FUNCTION_BLOCK FB_MotionStage_Test EXTENDS TcUnit.FB_TestSuite
VAR
    Expected: BOOL;
    Actual: BOOL;
END_VAR

TEST('FB_MotionStage_Test Dummy Test');
AssertEquals(Expected := Expected,
             Actual := Actual,
             Message := 'Error Message');
TEST_FINISHED();

END_FUNCTION_BLOCK

(* stored: Version 1.1.0.1, ProductVersion 3.1.4022.18
   POU FB_MotionStage_Test: Id {2872688d-0641-4c60-8808-69627b8ab29f}, SpecialFunc None *)
